TYPE tEncInState2 :
STRUCT	
	StatusInputA			: BIT;
	StatusInputB			: BIT;
	StatusExternLatch		: BIT;
	SyncError				: BIT;
	TxPdoToggle				: BIT;
END_STRUCT
END_TYPE

(* stored: Version 1.1.0.1, ProductVersion 3.1.4024.10
   DUT tEncInState2: Id {d680a987-6e3a-423d-bfcc-1e2f0197ef98} *)
